FUNCTION_BLOCK MockEnumerable IMPLEMENTS I_Enumerable
VAR
	enumerator : MockForwardEnumerator(FALSE,FALSE,FALSE,FALSE);
END_VAR

METHOD PUBLIC GetEnumerator : I_ForwardEnumerator
GetEnumerator := enumerator;
END_METHOD

END_FUNCTION_BLOCK

(* stored: Version 1.1.0.1, ProductVersion 3.1.4024.12
   POU MockEnumerable: Id {91f90a77-a44e-4ee3-8f71-353f56d1b688}, SpecialFunc None
   Method GetEnumerator: Id {3c2bf8e0-a457-4dd0-a532-1814fdd460da} *)
